// TIA Portal V18 export
// export: Created 2025-12-01T12:38:54.3039674Z, ExportSetting None, DisplayName Totally Integrated Automation Portal, DisplayVersion V18 Update 5, DisplayName TIA Portal Openness, DisplayVersion V18 Update 5, DisplayName TIA Portal Teamcenter Gateway, DisplayVersion V18, DisplayName TIA Portal Version Control Interface, DisplayVersion V18, DisplayName STEP 7 Professional, DisplayVersion V18 Update 5, DisplayName STEP 7 Safety, DisplayVersion V18, DisplayName WinCC Professional, DisplayVersion V18 Update 5
DATA_BLOCK "PartDataManage_Part3_DB"   // DB1503
// stored: InstanceOfName PartDataManage, InstanceOfType FB
"PartDataManage"
   // VAR_INPUT
   //    iReset : Bool;
   //    iScannerTrigger : Bool;
   //    iStringRecived : String;
   //    iMaterialType : String;
   //    iSaveToBuffer : Bool;
   //    iCodeType : Bool;
   //    iDecrementCnt : DInt;
   //    iDecrementTrigger : Bool;
   //    iBufferBoxes : Int;
   // END_VAR
   // VAR_IN_OUT
   //    ioMaterialActive : Bool;
   //    io_MaterialManage : "PartData_UDT";
   // END_VAR
   // VAR
   //    NO : Array[0..6] of Int;
   //    sString_MId : String;
   //    sKeyChar : Char;
   //    Puls : Array[0..20] of Bool;
   //    R_TRIG_MaterialActive { S7_SetPoint := 'True'} : R_TRIG;
   //    R_TRIG_ScannerTrigger { S7_SetPoint := 'True'} : R_TRIG;
   //    IEC_Timer_MaterialActive { S7_SetPoint := 'True'} : TON_TIME;
   //    R_TRIG_DecrementTrigger { S7_SetPoint := 'True'} : R_TRIG;
   //    "R_TRIG_PartQuality+1" { S7_SetPoint := 'True'} : R_TRIG;
   //    "R_TRIG_PartQuality-1" { S7_SetPoint := 'True'} : R_TRIG;
   //    R_TRIG_ClearCurrentBox { S7_SetPoint := 'True'} : R_TRIG;
   //    R_TRIG_ClearAllBox { S7_SetPoint := 'True'} : R_TRIG;
   //    R_TRIG_SaveToBuffer { S7_SetPoint := 'True'} : R_TRIG;
   //    Timer_PartQualityAckPB { S7_SetPoint := 'True'} : TON_TIME;
   // END_VAR
BEGIN
END_DATA_BLOCK
